PROGRAM Modbus
VAR
	fbModbusRtuMaster_PcCOM:ModbusRtuMaster_PcCOM;
	ChillerRead : ARRAY[0..10] OF WORD;
	ChillerWrite : ARRAY[0..10] OF WORD;

	bWrite: BOOL;
	bRead: BOOL;
	
	fbTON :TON;
	fbTONTrig : TON;
END_VAR

fbTON(IN:=NOT(fbTONTrig.Q), PT:= T#1S);
fbTONTrig(IN:=fbTON.Q, PT:= T#1s);


fbModbusRtuMaster_PcCOM.ReadRegs(
	UnitID:= 01, 
	Quantity:= 7, 
	MBAddr:= 16#0
, 
	cbLength:= SIZEOF(ChillerRead), 
	pMemoryAddr:= ADR(ChillerRead), 
	Execute:= fbTON.Q, 
	Timeout:= T#5S);
	
IO.ChillerTemperature := WORD_TO_REAL(ChillerRead[5]);
ChillerWrite[0] := REAL_TO_WORD(IO.ChillerTempSetpoint);	
	
fbModbusRtuMaster_PcCOM.WriteRegs(
	UnitID:= 01, 
	Quantity:= 1, 
	MBAddr:= 16#8, 
	cbLength:= SIZEOF(ChillerWrite), 
	pMemoryAddr:= ADR(ChillerWrite), 
	Execute:= NOT(fbTON.Q), 
	Timeout:= T#5S);

END_PROGRAM

(* stored: Version 1.1.0.1, ProductVersion 3.1.4024.9
   POU Modbus: Id {916482c7-f302-4872-b236-f0924dd81096}, SpecialFunc None *)
